PROGRAM Stn053_67_Stn232Merge
VAR
	{attribute 'TcLinkToOSO' := '.iBufferFull :=  <0,1,2>TIIB[N41S00 (AL1332)]^N41S03 (AL2341)^TxPDO^input byte 2'}	
	fbConvMerge: FB_ConvMerge;		
	{attribute 'TcLinkToOSO' := '<0,1,2>TIIB[N41S00 (AL1332)]^N41S03 (AL2341)^TxPDO^input byte 2'}
	iBufferFull AT %I*: BOOL;
END_VAR

//  This code instantiates a component that is implimented as a common function block
//    Note that I/O is linked directly to I/O variables inside the named instance

gStn053_67_Stn232Merge.MainHeartbeatOK := TRUE; // because this PLC is Main
gStn053_67_Stn232Merge.MainConvRunning :=  gConsumed_SafetyInterfaceConv.MtrRunning.Enc057Mtr01;
gStn053_67_Stn232Merge.MainInAuto := gStn053.CycleAuto;

gStn053_67_Stn232Merge.SpurHeartbeatOK := gConsumed_Stn232To053_OK;
gStn053_67_Stn232Merge.SpurConvRunning := gConsumed_Stn232To053.SpurConvRunning;
gStn053_67_Stn232Merge.SpurInAuto := gConsumed_Stn232To053.ScratchPad[0].2;

gStn232_30_MergeSpurPreStop.Available := gConsumed_Stn232To053.Available;


fbConvMerge(
	pStn := ADR(gStn053),
	pCmp := ADR(gStn053_67_Stn232Merge),
	pStateTraceBuffer := ADR(gStn053_StateTraceBuffer),
	pStateTraceFifo := ADR(gStn053_StateTraceFifo),
	pStats := ADR(gStn053_02_Stats),
	pMain := ADR(gStn053_66_Stn232MainMergePrestop),
	pSpur := ADR(gStn232_30_MergeSpurPreStop)		
);

gProduced_Stn053To232.Release := gStn232_30_MergeSpurPreStop.Release;
gProduced_Stn053To232.iBufferFull := iBufferFull;

END_PROGRAM

(* stored: Version 1.1.0.1, ProductVersion 3.1.4024.6
   POU Stn053_67_Stn232Merge: Id {a2a9988f-61ee-4acf-8e2c-7eced9bd8f15}, SpecialFunc None *)
